ABB RAPID module: Pickandplace.mod

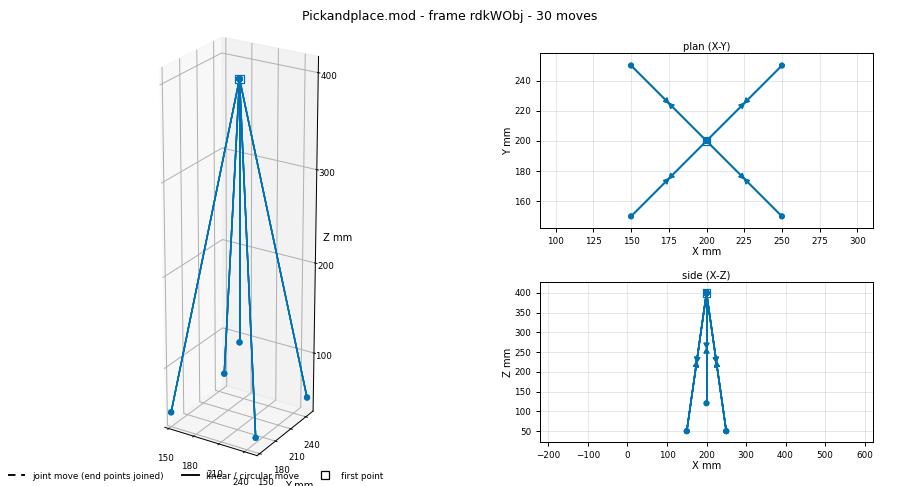
[picture p0: tool path of Pickandplace.mod in frame rdkWObj, 30 of 30 moves have a stored position in this frame; points joined in program order, loops and branches not executed]
MODULE MOD_Pickandplace

PERS wobjdata rdkWObj := [FALSE, TRUE, "", [[0,0,0],[1,0,0,0]],[[0,0,0],[1,0,0,0]]];
PERS tooldata rdkTool := [TRUE,[[0,0,0],[1,0,0,0]],[6.8,[0,0,15],[1,0,0,0],0,0,0.005]];
VAR speeddata rdkSpeed := [500,500,500,500];
VAR zonedata rdkZone := z0;
VAR extjoint rdkExtax := [9E9,9E9,9E9,9E9,9E9,9E9];

PROC main_RoboDK()
	Pickandplace;
	EXIT;
ENDPROC

PROC Pickandplace()
	!Program generated by RoboDK 2.4.0 for ABB IRB 1600-8/1.45 on 26/06/2016 15:07:59
	!Using nominal kinematics.
	var robtarget crt;
	crt := CRobT(\Tool:=rdkTool, \WObj:=rdkWObj);
	rdkExtax := crt.extax;
	ConfJ \On;
	ConfL \Off;
	rdkWObj.uframe:=[[0.000,0.000,0.000],[1.00000000,0.00000000,0.00000000,0.00000000]];
	rdkWObj.oframe:=[[631.624,-821.056,593.740],[1.00000000,0.00000000,0.00000000,0.00000000]];
	rdkTool.tframe:=[[125.000,0.000,100.000],[0.70710678,0.00000000,0.70710678,0.00000001]];
	MoveJ [[200.000,200.000,400.000],[0.00000000,0.00000000,-1.00000000,0.00000000],[-1,-1,0,1],rdkExtax], rdkSpeed, rdkZone, rdkTool, \WObj:=rdkWObj;
	MoveL [[200.000,200.000,120.711],[0.00000000,0.00000000,1.00000000,0.00000000],[-1,0,-1,2],rdkExtax], rdkSpeed, rdkZone, rdkTool, \WObj:=rdkWObj;
	!Attach to Tool
	AirValve_On;
	MoveL [[200.000,200.000,400.000],[0.00000000,0.00000000,-1.00000000,0.00000000],[-1,-1,0,1],rdkExtax], rdkSpeed, rdkZone, rdkTool, \WObj:=rdkWObj;
	rdkWObj.uframe:=[[0.000,0.000,0.000],[1.00000000,0.00000000,0.00000000,0.00000000]];
	rdkWObj.oframe:=[[681.663,630.034,534.204],[1.00000000,0.00000000,0.00000000,0.00000000]];
	MoveJ [[200.000,200.000,400.000],[0.00000000,0.00000000,-1.00000000,0.00000000],[-1,-1,0,1],rdkExtax], rdkSpeed, rdkZone, rdkTool, \WObj:=rdkWObj;
	MoveL [[150.000,150.000,50.000],[0.00000000,0.00000000,-1.00000000,0.00000000],[-1,-1,0,1],rdkExtax], rdkSpeed, rdkZone, rdkTool, \WObj:=rdkWObj;
	!Detach from Tool
	AirValve_Off;
	MoveL [[200.000,200.000,400.000],[0.00000000,0.00000000,-1.00000000,0.00000000],[-1,-1,0,1],rdkExtax], rdkSpeed, rdkZone, rdkTool, \WObj:=rdkWObj;
	rdkWObj.uframe:=[[0.000,0.000,0.000],[1.00000000,0.00000000,0.00000000,0.00000000]];
	rdkWObj.oframe:=[[631.624,-821.056,593.740],[1.00000000,0.00000000,0.00000000,0.00000000]];
	MoveJ [[200.000,200.000,400.000],[0.00000000,0.00000000,-1.00000000,0.00000000],[-1,-1,0,1],rdkExtax], rdkSpeed, rdkZone, rdkTool, \WObj:=rdkWObj;
	MoveL [[250.000,250.000,50.000],[0.00000000,0.00000000,1.00000000,0.00000000],[-1,1,-2,0],rdkExtax], rdkSpeed, rdkZone, rdkTool, \WObj:=rdkWObj;
	!Attach to Tool
	AirValve_On;
	MoveL [[200.000,200.000,400.000],[0.00000000,0.00000000,-1.00000000,0.00000000],[-1,-1,0,1],rdkExtax], rdkSpeed, rdkZone, rdkTool, \WObj:=rdkWObj;
	rdkWObj.uframe:=[[0.000,0.000,0.000],[1.00000000,0.00000000,0.00000000,0.00000000]];
	rdkWObj.oframe:=[[681.663,630.034,534.204],[1.00000000,0.00000000,0.00000000,0.00000000]];
	MoveJ [[200.000,200.000,400.000],[0.00000000,0.00000000,-1.00000000,0.00000000],[-1,-1,0,1],rdkExtax], rdkSpeed, rdkZone, rdkTool, \WObj:=rdkWObj;
	MoveL [[250.000,150.000,50.000],[0.00000000,0.00000000,1.00000000,0.00000000],[-1,1,-2,0],rdkExtax], rdkSpeed, rdkZone, rdkTool, \WObj:=rdkWObj;
	!Detach from Tool
	AirValve_Off;
	MoveL [[200.000,200.000,400.000],[0.00000000,0.00000000,-1.00000000,0.00000000],[-1,-1,0,1],rdkExtax], rdkSpeed, rdkZone, rdkTool, \WObj:=rdkWObj;
	rdkWObj.uframe:=[[0.000,0.000,0.000],[1.00000000,0.00000000,0.00000000,0.00000000]];
	rdkWObj.oframe:=[[631.624,-821.056,593.740],[1.00000000,0.00000000,0.00000000,0.00000000]];
	MoveJ [[200.000,200.000,400.000],[0.00000000,0.00000000,-1.00000000,0.00000000],[-1,-1,0,1],rdkExtax], rdkSpeed, rdkZone, rdkTool, \WObj:=rdkWObj;
	MoveL [[150.000,250.000,50.000],[0.00000000,0.00000000,1.00000000,0.00000000],[-1,1,-2,0],rdkExtax], rdkSpeed, rdkZone, rdkTool, \WObj:=rdkWObj;
	!Attach to Tool
	AirValve_On;
	MoveL [[200.000,200.000,400.000],[0.00000000,0.00000000,-1.00000000,0.00000000],[-1,-1,0,1],rdkExtax], rdkSpeed, rdkZone, rdkTool, \WObj:=rdkWObj;
	rdkWObj.uframe:=[[0.000,0.000,0.000],[1.00000000,0.00000000,0.00000000,0.00000000]];
	rdkWObj.oframe:=[[681.663,630.034,534.204],[1.00000000,0.00000000,0.00000000,0.00000000]];
	MoveJ [[200.000,200.000,400.000],[0.00000000,0.00000000,-1.00000000,0.00000000],[-1,-1,0,1],rdkExtax], rdkSpeed, rdkZone, rdkTool, \WObj:=rdkWObj;
	MoveL [[150.000,250.000,50.000],[0.00000000,0.00000000,1.00000000,0.00000000],[-1,1,-2,0],rdkExtax], rdkSpeed, rdkZone, rdkTool, \WObj:=rdkWObj;
	!Detach from Tool
	AirValve_Off;
	MoveL [[200.000,200.000,400.000],[0.00000000,0.00000000,-1.00000000,0.00000000],[-1,-1,0,1],rdkExtax], rdkSpeed, rdkZone, rdkTool, \WObj:=rdkWObj;
	rdkWObj.uframe:=[[0.000,0.000,0.000],[1.00000000,0.00000000,0.00000000,0.00000000]];
	rdkWObj.oframe:=[[631.624,-821.056,593.740],[1.00000000,0.00000000,0.00000000,0.00000000]];
	MoveJ [[200.000,200.000,400.000],[0.00000000,0.00000000,-1.00000000,0.00000000],[-1,-1,0,1],rdkExtax], rdkSpeed, rdkZone, rdkTool, \WObj:=rdkWObj;
	MoveL [[250.000,150.000,50.000],[0.00000000,0.00000000,1.00000000,0.00000000],[-1,1,-2,0],rdkExtax], rdkSpeed, rdkZone, rdkTool, \WObj:=rdkWObj;
	!Attach to Tool
	AirValve_On;
	MoveL [[200.000,200.000,400.000],[0.00000000,0.00000000,-1.00000000,0.00000000],[-1,-1,0,1],rdkExtax], rdkSpeed, rdkZone, rdkTool, \WObj:=rdkWObj;
	rdkWObj.uframe:=[[0.000,0.000,0.000],[1.00000000,0.00000000,0.00000000,0.00000000]];
	rdkWObj.oframe:=[[681.663,630.034,534.204],[1.00000000,0.00000000,0.00000000,0.00000000]];
	MoveJ [[200.000,200.000,400.000],[0.00000000,0.00000000,-1.00000000,0.00000000],[-1,-1,0,1],rdkExtax], rdkSpeed, rdkZone, rdkTool, \WObj:=rdkWObj;
	MoveL [[250.000,250.000,50.000],[0.00000000,0.00000000,1.00000000,0.00000000],[-1,1,-2,0],rdkExtax], rdkSpeed, rdkZone, rdkTool, \WObj:=rdkWObj;
	!Detach from Tool
	AirValve_Off;
	MoveL [[200.000,200.000,400.000],[0.00000000,0.00000000,-1.00000000,0.00000000],[-1,-1,0,1],rdkExtax], rdkSpeed, rdkZone, rdkTool, \WObj:=rdkWObj;
	rdkWObj.uframe:=[[0.000,0.000,0.000],[1.00000000,0.00000000,0.00000000,0.00000000]];
	rdkWObj.oframe:=[[631.624,-821.056,593.740],[1.00000000,0.00000000,0.00000000,0.00000000]];
	MoveJ [[200.000,200.000,400.000],[0.00000000,0.00000000,-1.00000000,0.00000000],[-1,-1,0,1],rdkExtax], rdkSpeed, rdkZone, rdkTool, \WObj:=rdkWObj;
	MoveL [[150.000,150.000,50.000],[0.00000000,0.00000000,-1.00000000,0.00000000],[-1,-1,0,1],rdkExtax], rdkSpeed, rdkZone, rdkTool, \WObj:=rdkWObj;
	!Attach to Tool
	AirValve_On;
	MoveL [[200.000,200.000,400.000],[0.00000000,0.00000000,-1.00000000,0.00000000],[-1,-1,0,1],rdkExtax], rdkSpeed, rdkZone, rdkTool, \WObj:=rdkWObj;
	rdkWObj.uframe:=[[0.000,0.000,0.000],[1.00000000,0.00000000,0.00000000,0.00000000]];
	rdkWObj.oframe:=[[681.663,630.034,534.204],[1.00000000,0.00000000,0.00000000,0.00000000]];
	MoveJ [[200.000,200.000,400.000],[0.00000000,0.00000000,-1.00000000,0.00000000],[-1,-1,0,1],rdkExtax], rdkSpeed, rdkZone, rdkTool, \WObj:=rdkWObj;
	MoveL [[200.000,200.000,120.711],[0.00000000,0.00000000,1.00000000,0.00000000],[-1,0,-1,2],rdkExtax], rdkSpeed, rdkZone, rdkTool, \WObj:=rdkWObj;
	!Detach from Tool
	AirValve_Off;
	MoveL [[200.000,200.000,400.000],[0.00000000,0.00000000,-1.00000000,0.00000000],[-1,-1,0,1],rdkExtax], rdkSpeed, rdkZone, rdkTool, \WObj:=rdkWObj;
	WaitTime \InPos, 5.000;
	Replaceobjects;
ENDPROC

PROC Replace objects()
	!Replace objects
ENDPROC

ENDMODULE
